TYPE "udtStanowiskoAssembly"
VERSION : 0.1
   STRUCT
      Config : Struct
         ID : Int;
         "Name" : String[20];
         HorlyRate : Real;
      END_STRUCT;
      Production : Struct
         State : Int;   // 0 - Gotowy. 1 - Montaż, 2 - Zakończono, 3 - Awaria
         OrderNo : Int;
         ProductNo : Int;
      END_STRUCT;
      "Time" : Struct
         TargetTime : Time;
         LastSec : UInt;
         RemainingSec : Int;
         RemainingStr : String[6];
         Blink : Bool;
      END_STRUCT;
      Commands : Struct
         Start : Struct
            Enable : Bool;
            State : Bool;
         END_STRUCT;
         FInish : Struct
            Enable : Bool;
            State : Bool;
         END_STRUCT;
         ReportFault : Struct
            Enable : Bool;
            State : Bool;
         END_STRUCT;
         AbortProcess : Struct
            Enable : Bool;
            State : Bool;
         END_STRUCT;
         FaultReason : Struct
            MissingPart : Bool;
            DamagedPart : Bool;
            PalletFault : Bool;
            WrongInstruction : Bool;
            SensorFault : Bool;
            Other : Bool;
         END_STRUCT;
      END_STRUCT;
      Sensors : Struct
         PalletPresent : Bool;
         RFID : Struct
            TagPresent : Bool;
            CmdRead : Bool;
            CmdWrite : Bool;
            Status : Bool;
            OrderNo : Int;
            ProductNo : Int;
         END_STRUCT;
      END_STRUCT;
      Stats : Struct
         DoneToday : Int;
         Efficiency : Int;
         ActudalPart : Int;
         Instruction : Int;
         Loaded : Bool;
      END_STRUCT;
      HMI : Struct
         Clear : Bool;   // Czyści licznik
         Container : Array[1..3] of Struct   // Tablica kontenerów
            value : Int;   // Ilość kontenerów 0 - 3
            Add : Struct   // Impuls na reczne dodanie
               Enable : Bool;
               Status : Bool;
            END_STRUCT;
            Subtract : Struct   // Impuls na reczne odejmowanie
               Enable : Bool;
               Status : Bool;
            END_STRUCT;
         END_STRUCT;
      END_STRUCT;
      MontazState : Int;
   END_STRUCT;

END_TYPE

DATA_BLOCK "DB_Data"
{ S7_Optimized_Access := 'FALSE' }
VERSION : 0.1
   STRUCT
      Stanowisko1 { S7_SetPoint := 'False'} : "udtStanowiskoAssembly";
      Stanowisko2 : "udtStanowiskoAssembly";
      Stanowisko3 : "udtStanowiskoAssembly";
      StanowiskoQC : Struct
         Config : Struct
            ID : Int;
            "Name" : String[20];
            HorlyRate : Real;
         END_STRUCT;
         Production : Struct
            State : Int;
            OrderNo : Int;
            ProductNo : Int;
         END_STRUCT;
         "Time" : Struct
            TargetTime : Time;
            LastSec : UInt;
            RemainingSec : Int;
            RemainingStr : String[6];
            Blink : Bool;
         END_STRUCT;
         Commands : Struct
            Start : Struct
               Enable : Bool;
               State : Bool;
            END_STRUCT;
            OK : Struct
               Enable : Bool;
               State : Bool;
            END_STRUCT;
            NOK : Struct
               Enable : Bool;
               State : Bool;
               NoBrick : Bool;
               WrongColour : Bool;
               Offset : Bool;
               Damage : Bool;
               WrongNumber : Bool;
               Other : Bool;
            END_STRUCT;
            ReportFault : Struct
               Enable : Bool;
               State : Bool;
            END_STRUCT;
         END_STRUCT;
         Sensors : Struct
            PalletPresent : Bool;
            RFID : Struct
               TagPresent : Bool;
               CmdRead : Bool;
               CmdWrite : Bool;
               Status : Bool;
               OrderNo : Int;
               ProductNo : Int;
            END_STRUCT;
         END_STRUCT;
         Stats : Struct
            DoneToday : Int;
            Efficiency : Int;
            ActudalPart : Int;
            Instruction : Int;
            Loaded : Bool;
            PartsOK : Int;
            PartsNOK : Int;
            PartsPercent : Int;
         END_STRUCT;
         HMI : Struct
            Clear : Bool;
            CameraStatus : Int;
         END_STRUCT;
         QualityState : Int;
         FaultReason : Struct
            Camera : Bool;
            NOK : Bool;
            PalletFault : Bool;
            RFID : Bool;
            SensorFault : Bool;
            Other : Bool;
         END_STRUCT;
         CameraControl : Struct
            bInit : Bool;
            bGetResult : Bool;
            bResetError : Bool;
            wynikOK : Bool;
            bReq : Bool;
            bTrigger : Bool;
            bZrobInspekcje : Bool;
            krok : Int;
            wynikOV : Array[0..5] of Bool;
            CameraStatus : Bool;
         END_STRUCT;
      END_STRUCT;
      ZlecenieIndex { S7_SetPoint := 'True'} : Array[0..3] of Int;
      DoneAllTime : Array[0..3] of Int;
   END_STRUCT;


BEGIN
   Stanowisko1.Production.State := 0;
   Stanowisko1.Production.OrderNo := 0;

END_DATA_BLOCK

ORGANIZATION_BLOCK "Kontenery"
TITLE = "Main Program Sweep (Cycle)"
{ S7_Optimized_Access := 'TRUE' }
VERSION : 0.1

BEGIN
	// ==========================================================================
	// Stanowisko 1
	// ==========================================================================
	//Tor 1
	IF "DB_Data".Stanowisko1.HMI.Container[1].value = 0 THEN
	    "DB_Data".Stanowisko1.HMI.Container[1].Subtract.Enable := FALSE;
	    "DB_Data".Stanowisko1.HMI.Container[1].Add.Enable := TRUE;
	END_IF;
	IF "DB_Data".Stanowisko1.HMI.Container[1].value = 1 OR "DB_Data".Stanowisko1.HMI.Container[1].value = 2 THEN
	    "DB_Data".Stanowisko1.HMI.Container[1].Subtract.Enable := TRUE;
	    "DB_Data".Stanowisko1.HMI.Container[1].Add.Enable := TRUE;
	END_IF;
	IF "DB_Data".Stanowisko1.HMI.Container[1].value = 3 THEN
	    "DB_Data".Stanowisko1.HMI.Container[1].Add.Enable := FALSE;
	END_IF;
	IF "DB_Data".Stanowisko1.HMI.Container[1].Subtract.Status THEN
	    "DB_Data".Stanowisko1.HMI.Container[1].value -= 1;
	    "DB_Data".Stanowisko1.HMI.Container[1].Subtract.Status := FALSE;
	END_IF;
	IF "DB_Data".Stanowisko1.HMI.Container[1].Add.Status THEN
	    "DB_Data".Stanowisko1.HMI.Container[1].value += 1;
	    "DB_Data".Stanowisko1.HMI.Container[1].Add.Status := FALSE;
	END_IF;

	//Tor 2
	IF "DB_Data".Stanowisko1.HMI.Container[2].value = 0 THEN
	    "DB_Data".Stanowisko1.HMI.Container[2].Subtract.Enable := FALSE;
	    "DB_Data".Stanowisko1.HMI.Container[2].Add.Enable := TRUE;
	END_IF;
	IF "DB_Data".Stanowisko1.HMI.Container[2].value = 1 OR "DB_Data".Stanowisko1.HMI.Container[2].value = 2 THEN
	    "DB_Data".Stanowisko1.HMI.Container[2].Subtract.Enable := TRUE;
	    "DB_Data".Stanowisko1.HMI.Container[2].Add.Enable := TRUE;
	END_IF;
	IF "DB_Data".Stanowisko1.HMI.Container[2].value = 3 THEN
	    "DB_Data".Stanowisko1.HMI.Container[2].Add.Enable := FALSE;
	END_IF;
	IF "DB_Data".Stanowisko1.HMI.Container[2].Subtract.Status THEN
	    "DB_Data".Stanowisko1.HMI.Container[2].value -= 1;
	    "DB_Data".Stanowisko1.HMI.Container[2].Subtract.Status := FALSE;
	END_IF;
	IF "DB_Data".Stanowisko1.HMI.Container[2].Add.Status THEN
	    "DB_Data".Stanowisko1.HMI.Container[2].value += 1;
	    "DB_Data".Stanowisko1.HMI.Container[2].Add.Status := FALSE;
	END_IF;

	//Tor 3
	IF "DB_Data".Stanowisko1.HMI.Container[3].value = 0 THEN
	    "DB_Data".Stanowisko1.HMI.Container[3].Subtract.Enable := FALSE;
	    "DB_Data".Stanowisko1.HMI.Container[3].Add.Enable := TRUE;
	END_IF;
	IF "DB_Data".Stanowisko1.HMI.Container[3].value = 1 OR "DB_Data".Stanowisko1.HMI.Container[3].value = 2 THEN
	    "DB_Data".Stanowisko1.HMI.Container[3].Subtract.Enable := TRUE;
	    "DB_Data".Stanowisko1.HMI.Container[3].Add.Enable := TRUE;
	END_IF;
	IF "DB_Data".Stanowisko1.HMI.Container[3].value = 3 THEN
	    "DB_Data".Stanowisko1.HMI.Container[3].Add.Enable := FALSE;
	END_IF;
	IF "DB_Data".Stanowisko1.HMI.Container[3].Subtract.Status THEN
	    "DB_Data".Stanowisko1.HMI.Container[3].value -= 1;
	    "DB_Data".Stanowisko1.HMI.Container[3].Subtract.Status := FALSE;
	END_IF;
	IF "DB_Data".Stanowisko1.HMI.Container[3].Add.Status THEN
	    "DB_Data".Stanowisko1.HMI.Container[3].value += 1;
	    "DB_Data".Stanowisko1.HMI.Container[3].Add.Status := FALSE;
	END_IF;

	// ==========================================================================
	// Stanowisko 2
	// ==========================================================================
	//Tor 1
	IF "DB_Data".Stanowisko2.HMI.Container[1].value = 0 THEN
	    "DB_Data".Stanowisko2.HMI.Container[1].Subtract.Enable := FALSE;
	    "DB_Data".Stanowisko2.HMI.Container[1].Add.Enable := TRUE;
	END_IF;
	IF "DB_Data".Stanowisko2.HMI.Container[1].value = 1 OR "DB_Data".Stanowisko2.HMI.Container[1].value = 2 THEN
	    "DB_Data".Stanowisko2.HMI.Container[1].Subtract.Enable := TRUE;
	    "DB_Data".Stanowisko2.HMI.Container[1].Add.Enable := TRUE;
	END_IF;
	IF "DB_Data".Stanowisko2.HMI.Container[1].value = 3 THEN
	    "DB_Data".Stanowisko2.HMI.Container[1].Add.Enable := FALSE;
	END_IF;
	IF "DB_Data".Stanowisko2.HMI.Container[1].Subtract.Status THEN
	    "DB_Data".Stanowisko2.HMI.Container[1].value -= 1;
	    "DB_Data".Stanowisko2.HMI.Container[1].Subtract.Status := FALSE;
	END_IF;
	IF "DB_Data".Stanowisko2.HMI.Container[1].Add.Status THEN
	    "DB_Data".Stanowisko2.HMI.Container[1].value += 1;
	    "DB_Data".Stanowisko2.HMI.Container[1].Add.Status := FALSE;
	END_IF;

	//Tor 2
	IF "DB_Data".Stanowisko2.HMI.Container[2].value = 0 THEN
	    "DB_Data".Stanowisko2.HMI.Container[2].Subtract.Enable := FALSE;
	    "DB_Data".Stanowisko2.HMI.Container[2].Add.Enable := TRUE;
	END_IF;
	IF "DB_Data".Stanowisko2.HMI.Container[2].value = 1 OR "DB_Data".Stanowisko2.HMI.Container[2].value = 2 THEN
	    "DB_Data".Stanowisko2.HMI.Container[2].Subtract.Enable := TRUE;
	    "DB_Data".Stanowisko2.HMI.Container[2].Add.Enable := TRUE;
	END_IF;
	IF "DB_Data".Stanowisko2.HMI.Container[2].value = 3 THEN
	    "DB_Data".Stanowisko2.HMI.Container[2].Add.Enable := FALSE;
	END_IF;
	IF "DB_Data".Stanowisko2.HMI.Container[2].Subtract.Status THEN
	    "DB_Data".Stanowisko2.HMI.Container[2].value -= 1;
	    "DB_Data".Stanowisko2.HMI.Container[2].Subtract.Status := FALSE;
	END_IF;
	IF "DB_Data".Stanowisko2.HMI.Container[2].Add.Status THEN
	    "DB_Data".Stanowisko2.HMI.Container[2].value += 1;
	    "DB_Data".Stanowisko2.HMI.Container[2].Add.Status := FALSE;
	END_IF;

	//Tor 3
	IF "DB_Data".Stanowisko2.HMI.Container[3].value = 0 THEN
	    "DB_Data".Stanowisko2.HMI.Container[3].Subtract.Enable := FALSE;
	    "DB_Data".Stanowisko2.HMI.Container[3].Add.Enable := TRUE;
	END_IF;
	IF "DB_Data".Stanowisko2.HMI.Container[3].value = 1 OR "DB_Data".Stanowisko2.HMI.Container[3].value = 2 THEN
	    "DB_Data".Stanowisko2.HMI.Container[3].Subtract.Enable := TRUE;
	    "DB_Data".Stanowisko2.HMI.Container[3].Add.Enable := TRUE;
	END_IF;
	IF "DB_Data".Stanowisko2.HMI.Container[3].value = 3 THEN
	    "DB_Data".Stanowisko2.HMI.Container[3].Add.Enable := FALSE;
	END_IF;
	IF "DB_Data".Stanowisko2.HMI.Container[3].Subtract.Status THEN
	    "DB_Data".Stanowisko2.HMI.Container[3].value -= 1;
	    "DB_Data".Stanowisko2.HMI.Container[3].Subtract.Status := FALSE;
	END_IF;
	IF "DB_Data".Stanowisko2.HMI.Container[3].Add.Status THEN
	    "DB_Data".Stanowisko2.HMI.Container[3].value += 1;
	    "DB_Data".Stanowisko2.HMI.Container[3].Add.Status := FALSE;
	END_IF;

	// ==========================================================================
	// Stanowisko 3
	// ==========================================================================
	//Tor 1
	IF "DB_Data".Stanowisko3.HMI.Container[1].value = 0 THEN
	    "DB_Data".Stanowisko3.HMI.Container[1].Subtract.Enable := FALSE;
	    "DB_Data".Stanowisko3.HMI.Container[1].Add.Enable := TRUE;
	END_IF;
	IF "DB_Data".Stanowisko3.HMI.Container[1].value = 1 OR "DB_Data".Stanowisko3.HMI.Container[1].value = 2 THEN
	    "DB_Data".Stanowisko3.HMI.Container[1].Subtract.Enable := TRUE;
	    "DB_Data".Stanowisko3.HMI.Container[1].Add.Enable := TRUE;
	END_IF;
	IF "DB_Data".Stanowisko3.HMI.Container[1].value = 3 THEN
	    "DB_Data".Stanowisko3.HMI.Container[1].Add.Enable := FALSE;
	END_IF;
	IF "DB_Data".Stanowisko3.HMI.Container[1].Subtract.Status THEN
	    "DB_Data".Stanowisko3.HMI.Container[1].value -= 1;
	    "DB_Data".Stanowisko3.HMI.Container[1].Subtract.Status := FALSE;
	END_IF;
	IF "DB_Data".Stanowisko3.HMI.Container[1].Add.Status THEN
	    "DB_Data".Stanowisko3.HMI.Container[1].value += 1;
	    "DB_Data".Stanowisko3.HMI.Container[1].Add.Status := FALSE;
	END_IF;

	//Tor 2
	IF "DB_Data".Stanowisko3.HMI.Container[2].value = 0 THEN
	    "DB_Data".Stanowisko3.HMI.Container[2].Subtract.Enable := FALSE;
	    "DB_Data".Stanowisko3.HMI.Container[2].Add.Enable := TRUE;
	END_IF;
	IF "DB_Data".Stanowisko3.HMI.Container[2].value = 1 OR "DB_Data".Stanowisko3.HMI.Container[2].value = 2 THEN
	    "DB_Data".Stanowisko3.HMI.Container[2].Subtract.Enable := TRUE;
	    "DB_Data".Stanowisko3.HMI.Container[2].Add.Enable := TRUE;
	END_IF;
	IF "DB_Data".Stanowisko3.HMI.Container[2].value = 3 THEN
	    "DB_Data".Stanowisko3.HMI.Container[2].Add.Enable := FALSE;
	END_IF;
	IF "DB_Data".Stanowisko3.HMI.Container[2].Subtract.Status THEN
	    "DB_Data".Stanowisko3.HMI.Container[2].value -= 1;
	    "DB_Data".Stanowisko3.HMI.Container[2].Subtract.Status := FALSE;
	END_IF;
	IF "DB_Data".Stanowisko3.HMI.Container[2].Add.Status THEN
	    "DB_Data".Stanowisko3.HMI.Container[2].value += 1;
	    "DB_Data".Stanowisko3.HMI.Container[2].Add.Status := FALSE;
	END_IF;

	//Tor 3
	IF "DB_Data".Stanowisko3.HMI.Container[3].value = 0 THEN
	    "DB_Data".Stanowisko3.HMI.Container[3].Subtract.Enable := FALSE;
	    "DB_Data".Stanowisko3.HMI.Container[3].Add.Enable := TRUE;
	END_IF;
	IF "DB_Data".Stanowisko3.HMI.Container[3].value = 1 OR "DB_Data".Stanowisko3.HMI.Container[3].value = 2 THEN
	    "DB_Data".Stanowisko3.HMI.Container[3].Subtract.Enable := TRUE;
	    "DB_Data".Stanowisko3.HMI.Container[3].Add.Enable := TRUE;
	END_IF;
	IF "DB_Data".Stanowisko3.HMI.Container[3].value = 3 THEN
	    "DB_Data".Stanowisko3.HMI.Container[3].Add.Enable := FALSE;
	END_IF;
	IF "DB_Data".Stanowisko3.HMI.Container[3].Subtract.Status THEN
	    "DB_Data".Stanowisko3.HMI.Container[3].value -= 1;
	    "DB_Data".Stanowisko3.HMI.Container[3].Subtract.Status := FALSE;
	END_IF;
	IF "DB_Data".Stanowisko3.HMI.Container[3].Add.Status THEN
	    "DB_Data".Stanowisko3.HMI.Container[3].value += 1;
	    "DB_Data".Stanowisko3.HMI.Container[3].Add.Status := FALSE;
	END_IF;
END_ORGANIZATION_BLOCK

